// TIA Portal V17 export
// export: Created 2025-03-10T12:18:03.3825103Z, ExportSetting WithDefaults, DisplayName Totally Integrated Automation Portal, DisplayVersion V17 Update 8, DisplayName TIA Portal Openness, DisplayVersion V17 Update 8, DisplayName TIA Portal Version Control Interface, DisplayVersion V17, DisplayName SINAMICS Startdrive Advanced, DisplayVersion V17 SP2, DisplayName SINAMICS Startdrive G110M, G120, G120C, G120D, G120P, G115D, DisplayVersion V17 SP2, DisplayName SINAMICS Startdrive G130, G150, S120, S150, SINAMICS MV, S210, DisplayVersion V17 SP2, DisplayName STEP 7 Professional, DisplayVersion V17 Update 8, DisplayName SINUMERIK ONE STEP 7 Toolbox, DisplayVersion V17 Update 12, DisplayName SINUMERIK 840D sl STEP 7 Toolbox, DisplayVersion V17 Update 12, DisplayName STEP 7 Safety, DisplayVersion V17 Update 6, DisplayName WinCC Advanced, DisplayVersion V17 Update 8
TYPE "MR_J4_Aux_Control"
// stored: IsFailsafeCompliant false
   STRUCT
      Aux_Input : Struct
         SVON : Bool;
         SETUP : Bool;
         Jog_P : Bool;
         Jog_N : Bool;
         Reset : Bool;
         Hold : Bool;
         FLGTH : Bool;
         Speed_Restr : Bool;
         Start_Flag : Bool;
         Fly_Change : Bool;
         Continuous_Step : Bool;
      END_STRUCT;
      Aux_Output : Struct
         Svre : Bool;
         Seton : Bool;
         Busy : Bool;
         Inp : Bool;
         TLO : Bool;
         New_step_Ack : Bool;
         ILA : Bool;
         Warning : Bool;
         Alarm : Bool;
         Alarm_Bateria : Bool;
         Alarm_S_ABS : Bool;
         Voltage_Enable : Bool;
         LSN : Bool;
         LSP : Bool;
         Dog : Bool;
         STO1 : Bool;
         STO2 : Bool;
         Step_Actual : UInt;
         Pos_actual : DInt;
         Speed_Actual : Int;
         Par_Actual : Int;
         Pos_Pedida : DInt;
         Modo_Trabajo : Byte := 0;
         Alarma_Actual : DWord;
         Temperature_Encoder : DInt;
         Bus_Voltage : DInt;
         Efective_load_Ratio : DInt;
         Regenerative_load_Ratio : DInt;
      END_STRUCT;
      Aux_Param_Config : Struct
         Paso_Vuelta : UInt;
         "Velocidad maxima" : Int;
         Ac_DC_maxima : Int;
         Jog_speed : UInt;
         Jog_AC_DC : UInt;
         Torque_max_speed : Int;
         Torque_Max_TQ : Int;
         Torque_SLope_TQ : Int;
      END_STRUCT;
   END_STRUCT;
END_TYPE
